TYPE Read_BD_Values_To_PC_Struct :
UNION
	S_BDValues_To_PC:S_BDValues_To_PC_Struct;
END_UNION
END_TYPE

(* stored: Version 1.1.0.1, ProductVersion 3.1.4024.16
   DUT Read_BD_Values_To_PC_Struct: Id {d50f65be-a363-4d42-a051-c80706fe3a2a} *)
